{attribute 'qualified_only'}
{attribute 'strict'}
{attribute 'to_string'}
TYPE E_EventLoggerListenerState :
(	 
	eIdle := 0,
	eInit:= 1, 
	eListening:= 10, 
	eRetrieveTexts:= 20,
	eSortEvents := 30,
	eDone := 100,
	eError := -1
);
END_TYPE
//  eError = '-1'

(* stored: Version 1.1.0.1, ProductVersion 3.1.4024.12
   EnumerationTextList E_EventLoggerListenerState: Id {deae15e8-0c4a-4e95-a43c-a59572bbb9f7} *)
